// TIA Portal V19 export
FUNCTION_BLOCK "F_Zone21_FB"   // FB172, F_LAD
TITLE = SAFETY ZONE 21 - AREA 03 (ACCOPPIAMENTO)
// stored: Access Published
   VAR
      D19 : "Door_FB";
      D20 : "Door_FB";
      D21 : "Door_FB";
      FNS : "ForceNormalStop";
      F_Sinamics_Trasporto : "FDevice_Sinamics_FB";
      F_Sinamics_Ribaltatore : "FDevice_Sinamics_FB";
      F_Sinamics_Spintore : "FDevice_Sinamics_FB";
      F_Contactor_CambioFormato_Bordatrice { ExternalAccessible := 'False'; ExternalVisible := 'False'; ExternalWritable := 'False'} : "FDevice_Contactor_FB";
      F_Sinamics_Bordatrice : "FDevice_Sinamics_FB";
      F_SafetyValve_Air_A0301_A0302 : "FDevice_Valve_FB";
   END_VAR
   VAR_TEMP
      DoorNormalStop : Bool;
      DoorSafeStop : Bool;
      Door_Ok : Bool;
      FDBK : Bool;
   END_VAR
BEGIN

REGION Network 1: < < < < < < < < < < DOOR > > > > > > > > > >
END_REGION

REGION Network 2: Zone Entry enable
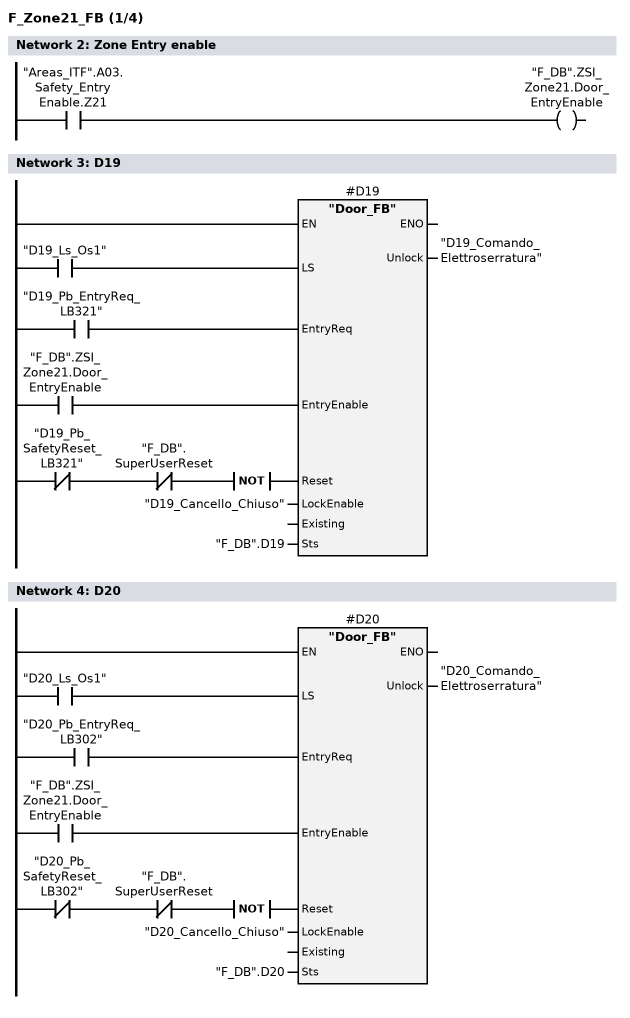
   RUNG wire#powerrail
      Contact( "Areas_ITF".A03.Safety_EntryEnable.Z21 )
      Coil( "F_DB".ZSI_Zone21.Door_EntryEnable )
   END_RUNG
   // the same network as SCL:
   "F_DB".ZSI_Zone21.Door_EntryEnable := "Areas_ITF".A03.Safety_EntryEnable.Z21;
END_REGION

REGION Network 3: D19
   RUNG wire#powerrail
      #D19(LS := wire#w1, EntryReq := wire#w2, EntryEnable := wire#w3, Reset := wire#w4, LockEnable := "D19_Cancello_Chiuso", Existing :=, Sts := "F_DB".D19, Unlock => "D19_Comando_Elettroserratura")
   END_RUNG
   RUNG wire#powerrail
      Contact( "D19_Ls_Os1" )
   END_RUNG wire#w1
   RUNG wire#powerrail
      Contact( "D19_Pb_EntryReq_LB321" )
   END_RUNG wire#w2
   RUNG wire#powerrail
      Contact( "F_DB".ZSI_Zone21.Door_EntryEnable )
   END_RUNG wire#w3
   RUNG wire#powerrail
      I_Contact( "D19_Pb_SafetyReset_LB321" )
      I_Contact( "F_DB".SuperUserReset )
      Not()
   END_RUNG wire#w4
   // the same network as SCL:
   #D19(LS := "D19_Ls_Os1",   // "Door_FB"
        EntryReq := "D19_Pb_EntryReq_LB321",
        EntryEnable := "F_DB".ZSI_Zone21.Door_EntryEnable,
        Reset := NOT (NOT "D19_Pb_SafetyReset_LB321" AND NOT "F_DB".SuperUserReset),
        LockEnable := "D19_Cancello_Chiuso",
        Sts := "F_DB".D19,
        Unlock => "D19_Comando_Elettroserratura");
END_REGION

REGION Network 4: D20
   RUNG wire#powerrail
      #D20(LS := wire#w1, EntryReq := wire#w2, EntryEnable := wire#w3, Reset := wire#w4, LockEnable := "D20_Cancello_Chiuso", Existing :=, Sts := "F_DB".D20, Unlock => "D20_Comando_Elettroserratura")
   END_RUNG
   RUNG wire#powerrail
      Contact( "D20_Ls_Os1" )
   END_RUNG wire#w1
   RUNG wire#powerrail
      Contact( "D20_Pb_EntryReq_LB302" )
   END_RUNG wire#w2
   RUNG wire#powerrail
      Contact( "F_DB".ZSI_Zone21.Door_EntryEnable )
   END_RUNG wire#w3
   RUNG wire#powerrail
      I_Contact( "D20_Pb_SafetyReset_LB302" )
      I_Contact( "F_DB".SuperUserReset )
      Not()
   END_RUNG wire#w4
   // the same network as SCL:
   #D20(LS := "D20_Ls_Os1",   // "Door_FB"
        EntryReq := "D20_Pb_EntryReq_LB302",
        EntryEnable := "F_DB".ZSI_Zone21.Door_EntryEnable,
        Reset := NOT (NOT "D20_Pb_SafetyReset_LB302" AND NOT "F_DB".SuperUserReset),
        LockEnable := "D20_Cancello_Chiuso",
        Sts := "F_DB".D20,
        Unlock => "D20_Comando_Elettroserratura");
END_REGION

REGION Network 5: D21
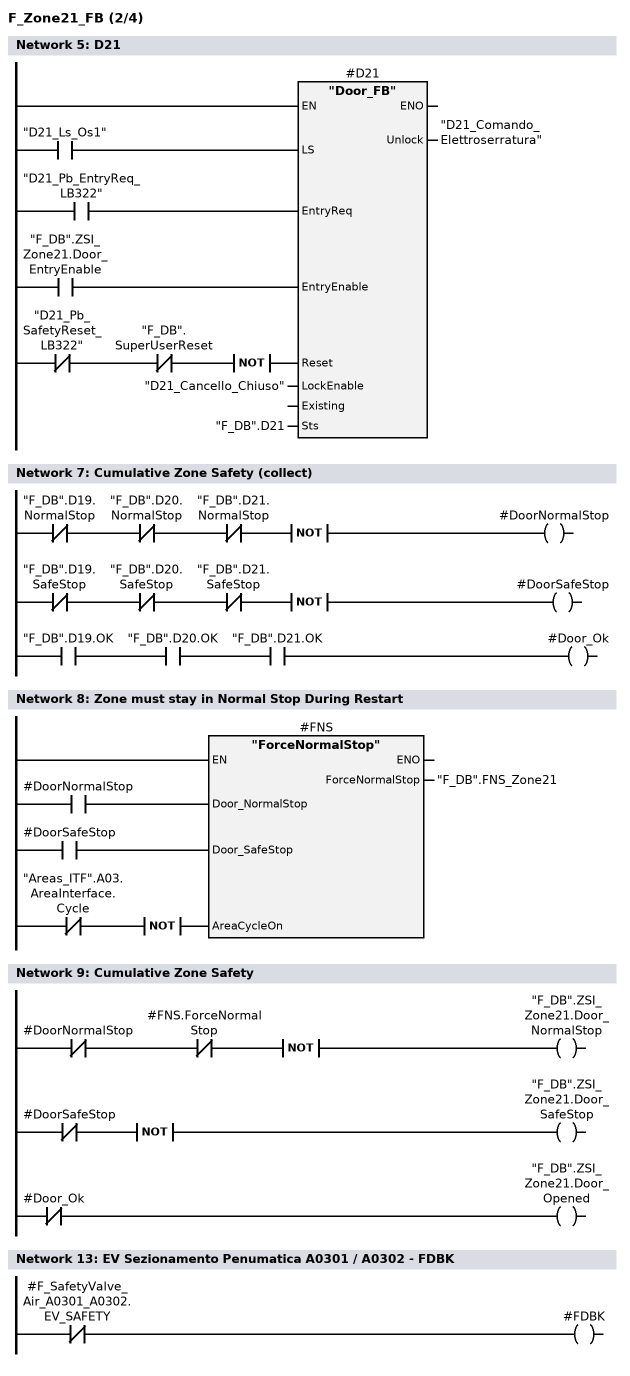
   RUNG wire#powerrail
      #D21(LS := wire#w1, EntryReq := wire#w2, EntryEnable := wire#w3, Reset := wire#w4, LockEnable := "D21_Cancello_Chiuso", Existing :=, Sts := "F_DB".D21, Unlock => "D21_Comando_Elettroserratura")
   END_RUNG
   RUNG wire#powerrail
      Contact( "D21_Ls_Os1" )
   END_RUNG wire#w1
   RUNG wire#powerrail
      Contact( "D21_Pb_EntryReq_LB322" )
   END_RUNG wire#w2
   RUNG wire#powerrail
      Contact( "F_DB".ZSI_Zone21.Door_EntryEnable )
   END_RUNG wire#w3
   RUNG wire#powerrail
      I_Contact( "D21_Pb_SafetyReset_LB322" )
      I_Contact( "F_DB".SuperUserReset )
      Not()
   END_RUNG wire#w4
   // the same network as SCL:
   #D21(LS := "D21_Ls_Os1",   // "Door_FB"
        EntryReq := "D21_Pb_EntryReq_LB322",
        EntryEnable := "F_DB".ZSI_Zone21.Door_EntryEnable,
        Reset := NOT (NOT "D21_Pb_SafetyReset_LB322" AND NOT "F_DB".SuperUserReset),
        LockEnable := "D21_Cancello_Chiuso",
        Sts := "F_DB".D21,
        Unlock => "D21_Comando_Elettroserratura");
END_REGION

REGION Network 6: < < < < < < < < < < ZONE SAFETY INTERFACE > > > > > > > > > >
END_REGION

REGION Network 7: Cumulative Zone Safety (collect)
   RUNG wire#powerrail
      I_Contact( "F_DB".D19.NormalStop )
      I_Contact( "F_DB".D20.NormalStop )
      I_Contact( "F_DB".D21.NormalStop )
      Not()
      Coil( #DoorNormalStop )
   END_RUNG
   RUNG wire#powerrail
      I_Contact( "F_DB".D19.SafeStop )
      I_Contact( "F_DB".D20.SafeStop )
      I_Contact( "F_DB".D21.SafeStop )
      Not()
      Coil( #DoorSafeStop )
   END_RUNG
   RUNG wire#powerrail
      Contact( "F_DB".D19.OK )
      Contact( "F_DB".D20.OK )
      Contact( "F_DB".D21.OK )
      Coil( #Door_Ok )
   END_RUNG
   // the same network as SCL:
   #DoorNormalStop := NOT (NOT "F_DB".D19.NormalStop AND NOT "F_DB".D20.NormalStop AND NOT "F_DB".D21.NormalStop);
   #DoorSafeStop := NOT (NOT "F_DB".D19.SafeStop AND NOT "F_DB".D20.SafeStop AND NOT "F_DB".D21.SafeStop);
   #Door_Ok := "F_DB".D19.OK AND "F_DB".D20.OK AND "F_DB".D21.OK;
END_REGION

REGION Network 8: Zone must stay in Normal Stop During Restart
   RUNG wire#powerrail
      #FNS(Door_NormalStop := wire#w1, Door_SafeStop := wire#w2, AreaCycleOn := wire#w3, ForceNormalStop => "F_DB".FNS_Zone21)
   END_RUNG
   RUNG wire#powerrail
      Contact( #DoorNormalStop )
   END_RUNG wire#w1
   RUNG wire#powerrail
      Contact( #DoorSafeStop )
   END_RUNG wire#w2
   RUNG wire#powerrail
      I_Contact( "Areas_ITF".A03.AreaInterface.Cycle )
      Not()
   END_RUNG wire#w3
   // the same network as SCL:
   #FNS(Door_NormalStop := #DoorNormalStop,   // "ForceNormalStop"
        Door_SafeStop := #DoorSafeStop,
        AreaCycleOn := NOT (NOT "Areas_ITF".A03.AreaInterface.Cycle),
        ForceNormalStop => "F_DB".FNS_Zone21);
END_REGION

REGION Network 9: Cumulative Zone Safety
   RUNG wire#powerrail
      I_Contact( #DoorNormalStop )
      I_Contact( #FNS.ForceNormalStop )
      Not()
      Coil( "F_DB".ZSI_Zone21.Door_NormalStop )
   END_RUNG
   RUNG wire#powerrail
      I_Contact( #DoorSafeStop )
      Not()
      Coil( "F_DB".ZSI_Zone21.Door_SafeStop )
   END_RUNG
   RUNG wire#powerrail
      I_Contact( #Door_Ok )
      Coil( "F_DB".ZSI_Zone21.Door_Opened )
   END_RUNG
   // the same network as SCL:
   "F_DB".ZSI_Zone21.Door_NormalStop := NOT (NOT #DoorNormalStop AND NOT #FNS.ForceNormalStop);
   "F_DB".ZSI_Zone21.Door_SafeStop := NOT (NOT #DoorSafeStop);
   "F_DB".ZSI_Zone21.Door_Opened := NOT #Door_Ok;
END_REGION

REGION Network 10: >
END_REGION

REGION Network 11: >
END_REGION

REGION Network 12: < < < < < < < < < < DEVICES SAFETY VALVES > > > > > > > > > >
END_REGION

REGION Network 13: EV Sezionamento Penumatica A0301 / A0302 - FDBK
   RUNG wire#powerrail
      I_Contact( #F_SafetyValve_Air_A0301_A0302.EV_SAFETY )
      Coil( #FDBK )
   END_RUNG
   // the same network as SCL:
   #FDBK := NOT #F_SafetyValve_Air_A0301_A0302.EV_SAFETY;
END_REGION

REGION Network 14: EV Sezionamento Pneumatica A0301 (Ribaltamento) + A0302 ingresso (bordatrice)
   // VALVOLA TAGLIATA SOLO DA EMERGENZA
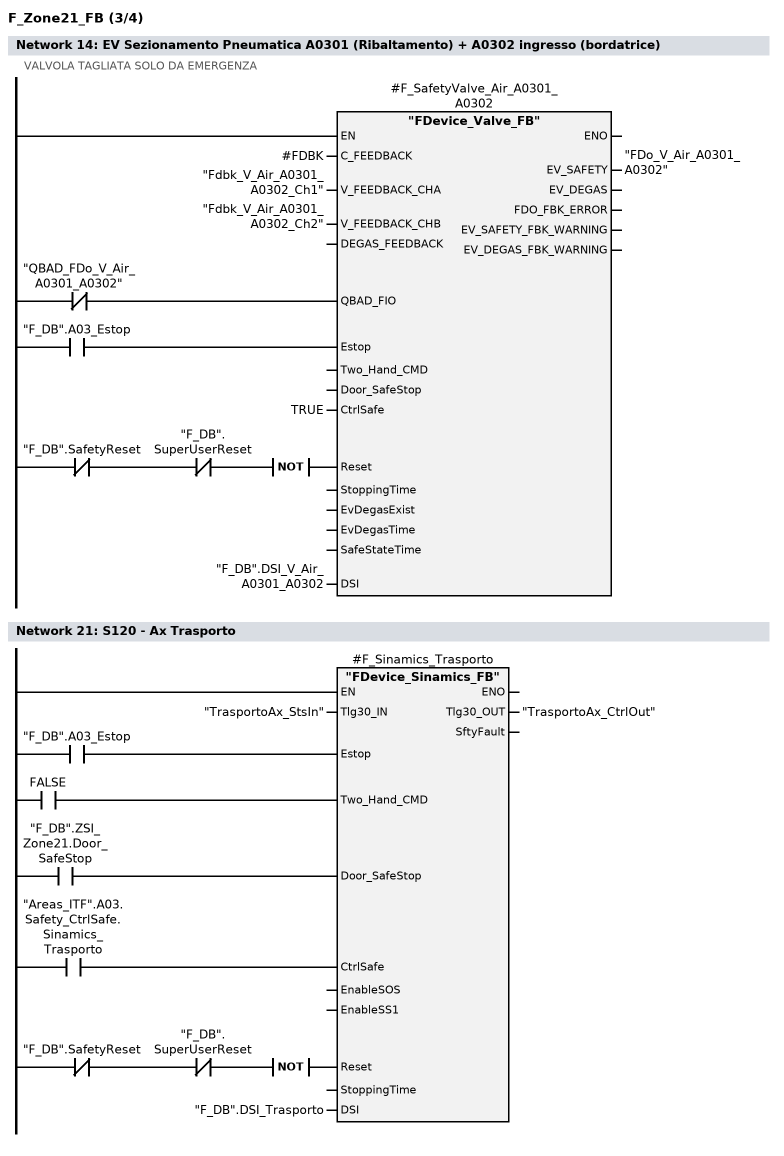
   RUNG wire#powerrail
      #F_SafetyValve_Air_A0301_A0302(QBAD_FIO := wire#w1, Estop := wire#w2, Reset := wire#w3, C_FEEDBACK := #FDBK, V_FEEDBACK_CHA := "Fdbk_V_Air_A0301_A0302_Ch1", V_FEEDBACK_CHB := "Fdbk_V_Air_A0301_A0302_Ch2", DEGAS_FEEDBACK :=, Two_Hand_CMD :=, Door_SafeStop :=, CtrlSafe := TRUE, StoppingTime :=, EvDegasExist :=, EvDegasTime :=, SafeStateTime :=, DSI := "F_DB".DSI_V_Air_A0301_A0302, EV_SAFETY => "FDo_V_Air_A0301_A0302", EV_DEGAS =>, FDO_FBK_ERROR =>, EV_SAFETY_FBK_WARNING =>, EV_DEGAS_FBK_WARNING =>)
   END_RUNG
   RUNG wire#powerrail
      I_Contact( "QBAD_FDo_V_Air_A0301_A0302" )
   END_RUNG wire#w1
   RUNG wire#powerrail
      Contact( "F_DB".A03_Estop )
   END_RUNG wire#w2
   RUNG wire#powerrail
      I_Contact( "F_DB".SafetyReset )
      I_Contact( "F_DB".SuperUserReset )
      Not()
   END_RUNG wire#w3
   // the same network as SCL:
   #F_SafetyValve_Air_A0301_A0302(C_FEEDBACK := #FDBK,   // "FDevice_Valve_FB"
                           V_FEEDBACK_CHA := "Fdbk_V_Air_A0301_A0302_Ch1",
                           V_FEEDBACK_CHB := "Fdbk_V_Air_A0301_A0302_Ch2",
                           QBAD_FIO := NOT "QBAD_FDo_V_Air_A0301_A0302",
                           Estop := "F_DB".A03_Estop,
                           CtrlSafe := TRUE,
                           Reset := NOT (NOT "F_DB".SafetyReset AND NOT "F_DB".SuperUserReset),
                           DSI := "F_DB".DSI_V_Air_A0301_A0302,
                           EV_SAFETY => "FDo_V_Air_A0301_A0302");
END_REGION

REGION Network 15: >
END_REGION

REGION Network 16: >
END_REGION

REGION Network 17: < < < < < < < < < < DEVICES CONTACTORS > > > > > > > > > >
END_REGION

REGION Network 18: >
END_REGION

REGION Network 19: >
END_REGION

REGION Network 20: < < < < < < < < < < DEVICES S120 > > > > > > > > > >
END_REGION

REGION Network 21: S120 - Ax Trasporto
   RUNG wire#powerrail
      #F_Sinamics_Trasporto(Estop := wire#w1, Two_Hand_CMD := wire#w2, Door_SafeStop := wire#w3, CtrlSafe := wire#w4, Reset := wire#w5, Tlg30_IN := "TrasportoAx_StsIn", EnableSOS :=, EnableSS1 :=, StoppingTime :=, DSI := "F_DB".DSI_Trasporto, Tlg30_OUT => "TrasportoAx_CtrlOut", SftyFault =>)
   END_RUNG
   RUNG wire#powerrail
      Contact( "F_DB".A03_Estop )
   END_RUNG wire#w1
   RUNG wire#powerrail
      Contact( FALSE )
   END_RUNG wire#w2
   RUNG wire#powerrail
      Contact( "F_DB".ZSI_Zone21.Door_SafeStop )
   END_RUNG wire#w3
   RUNG wire#powerrail
      Contact( "Areas_ITF".A03.Safety_CtrlSafe.Sinamics_Trasporto )
   END_RUNG wire#w4
   RUNG wire#powerrail
      I_Contact( "F_DB".SafetyReset )
      I_Contact( "F_DB".SuperUserReset )
      Not()
   END_RUNG wire#w5
   // the same network as SCL:
   #F_Sinamics_Trasporto(Tlg30_IN := "TrasportoAx_StsIn",   // "FDevice_Sinamics_FB"
                         Estop := "F_DB".A03_Estop,
                         Two_Hand_CMD := FALSE,
                         Door_SafeStop := "F_DB".ZSI_Zone21.Door_SafeStop,
                         CtrlSafe := "Areas_ITF".A03.Safety_CtrlSafe.Sinamics_Trasporto,
                         Reset := NOT (NOT "F_DB".SafetyReset AND NOT "F_DB".SuperUserReset),
                         DSI := "F_DB".DSI_Trasporto,
                         Tlg30_OUT => "TrasportoAx_CtrlOut");
END_REGION

REGION Network 22: S120 - Ax Ribaltatore
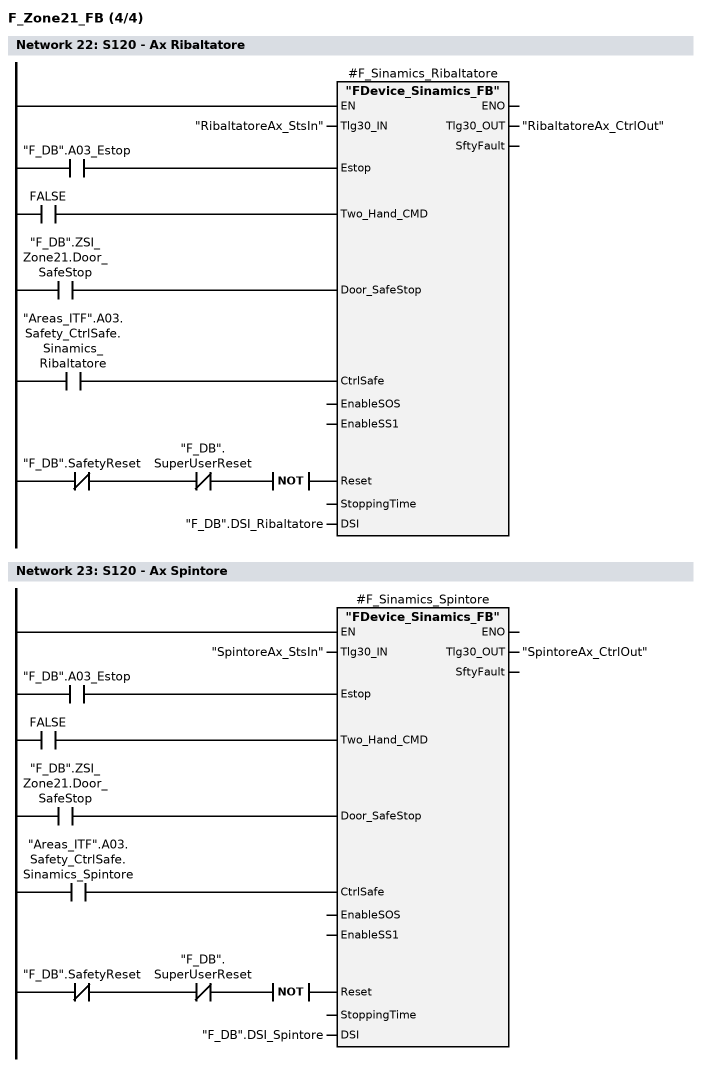
   RUNG wire#powerrail
      #F_Sinamics_Ribaltatore(Estop := wire#w1, Two_Hand_CMD := wire#w2, Door_SafeStop := wire#w3, CtrlSafe := wire#w4, Reset := wire#w5, Tlg30_IN := "RibaltatoreAx_StsIn", EnableSOS :=, EnableSS1 :=, StoppingTime :=, DSI := "F_DB".DSI_Ribaltatore, Tlg30_OUT => "RibaltatoreAx_CtrlOut", SftyFault =>)
   END_RUNG
   RUNG wire#powerrail
      Contact( "F_DB".A03_Estop )
   END_RUNG wire#w1
   RUNG wire#powerrail
      Contact( FALSE )
   END_RUNG wire#w2
   RUNG wire#powerrail
      Contact( "F_DB".ZSI_Zone21.Door_SafeStop )
   END_RUNG wire#w3
   RUNG wire#powerrail
      Contact( "Areas_ITF".A03.Safety_CtrlSafe.Sinamics_Ribaltatore )
   END_RUNG wire#w4
   RUNG wire#powerrail
      I_Contact( "F_DB".SafetyReset )
      I_Contact( "F_DB".SuperUserReset )
      Not()
   END_RUNG wire#w5
   // the same network as SCL:
   #F_Sinamics_Ribaltatore(Tlg30_IN := "RibaltatoreAx_StsIn",   // "FDevice_Sinamics_FB"
                           Estop := "F_DB".A03_Estop,
                           Two_Hand_CMD := FALSE,
                           Door_SafeStop := "F_DB".ZSI_Zone21.Door_SafeStop,
                           CtrlSafe := "Areas_ITF".A03.Safety_CtrlSafe.Sinamics_Ribaltatore,
                           Reset := NOT (NOT "F_DB".SafetyReset AND NOT "F_DB".SuperUserReset),
                           DSI := "F_DB".DSI_Ribaltatore,
                           Tlg30_OUT => "RibaltatoreAx_CtrlOut");
END_REGION

REGION Network 23: S120 - Ax Spintore
   RUNG wire#powerrail
      #F_Sinamics_Spintore(Estop := wire#w1, Two_Hand_CMD := wire#w2, Door_SafeStop := wire#w3, CtrlSafe := wire#w4, Reset := wire#w5, Tlg30_IN := "SpintoreAx_StsIn", EnableSOS :=, EnableSS1 :=, StoppingTime :=, DSI := "F_DB".DSI_Spintore, Tlg30_OUT => "SpintoreAx_CtrlOut", SftyFault =>)
   END_RUNG
   RUNG wire#powerrail
      Contact( "F_DB".A03_Estop )
   END_RUNG wire#w1
   RUNG wire#powerrail
      Contact( FALSE )
   END_RUNG wire#w2
   RUNG wire#powerrail
      Contact( "F_DB".ZSI_Zone21.Door_SafeStop )
   END_RUNG wire#w3
   RUNG wire#powerrail
      Contact( "Areas_ITF".A03.Safety_CtrlSafe.Sinamics_Spintore )
   END_RUNG wire#w4
   RUNG wire#powerrail
      I_Contact( "F_DB".SafetyReset )
      I_Contact( "F_DB".SuperUserReset )
      Not()
   END_RUNG wire#w5
   // the same network as SCL:
   #F_Sinamics_Spintore(Tlg30_IN := "SpintoreAx_StsIn",   // "FDevice_Sinamics_FB"
                        Estop := "F_DB".A03_Estop,
                        Two_Hand_CMD := FALSE,
                        Door_SafeStop := "F_DB".ZSI_Zone21.Door_SafeStop,
                        CtrlSafe := "Areas_ITF".A03.Safety_CtrlSafe.Sinamics_Spintore,
                        Reset := NOT (NOT "F_DB".SafetyReset AND NOT "F_DB".SuperUserReset),
                        DSI := "F_DB".DSI_Spintore,
                        Tlg30_OUT => "SpintoreAx_CtrlOut");
END_REGION

REGION Network 24: >
END_REGION

REGION Network 25: >
END_REGION
END_FUNCTION_BLOCK
